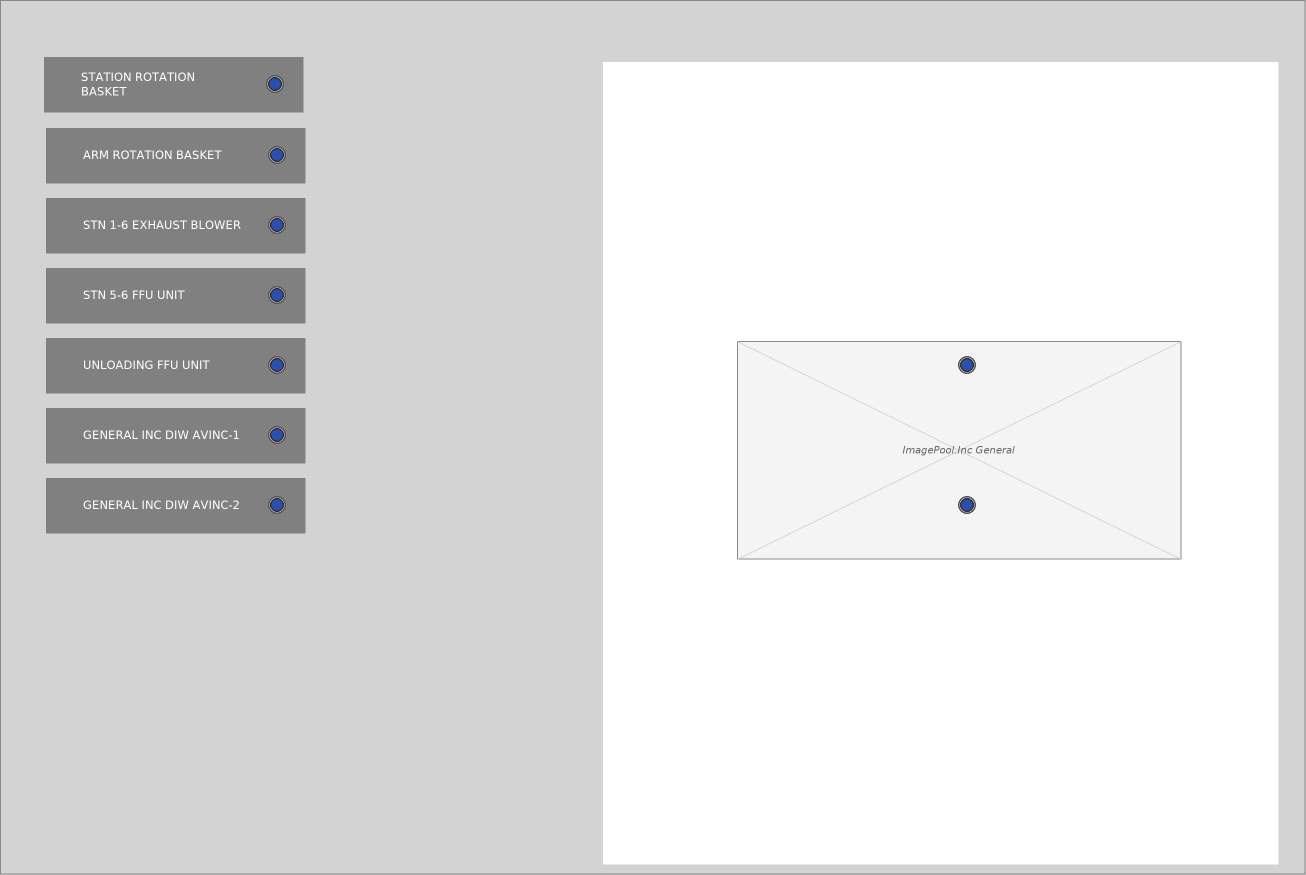
VISUALIZATION Auto_General  // 1306x875
    Rectangle (0,0 1306x875)
    Rectangle (603,62 675x802)
    RoundedRectangle (44,57 259x55)
    Label (78,71 176x27), "STATION ROTATION BASKET"
    Lamp1 (265,74 20x20), variable: ARdsMAP_HmiVariableGeneral.bStnRotationRotaryBarrel_IND, style: Lamp-Lamp1-Blue
    RoundedRectangle (46,198 259x55)
    Label (80,217 178x16), "STN 1-6 EXHAUST BLOWER"
    Lamp1 (267,215 20x20), variable: ARdsMAP_HmiVariableGeneral.bExhaustBlower_IND, style: Lamp-Lamp1-Blue
    Image (737,341 444x218), image: ImagePool.Inc General
    RoundedRectangle (46,408 259x55)
    Label (80,427 176x16), "GENERAL INC DIW AVINC-1"
    Lamp1 (267,425 20x20), variable: ARdsMAP_HmiVariableGeneral.bGeneralIncValve01_IND, style: Lamp-Lamp1-Blue
    RoundedRectangle (46,478 259x55)
    Label (80,497 178x16), "GENERAL INC DIW AVINC-2"
    Lamp1 (267,495 20x20), variable: ARdsMAP_HmiVariableGeneral.bGeneralIncValve02_IND, style: Lamp-Lamp1-Blue
    RoundedRectangle (46,128 259x55)
    Label (80,147 176x16), "ARM ROTATION BASKET"
    Lamp1 (267,145 20x20), variable: ARdsMAP_HmiVariableGeneral.bRobotRotationRotaryBarrel_IND, style: Lamp-Lamp1-Blue
    Lamp1 (957,355 20x20), variable: ARdsMAP_HmiVariableGeneral.bGeneralIncValve01_IND, style: Lamp-Lamp1-Blue
    Lamp1 (957,495 20x20), variable: ARdsMAP_HmiVariableGeneral.bGeneralIncValve02_IND, style: Lamp-Lamp1-Blue
    RoundedRectangle (46,268 259x55)
    Label (80,287 178x16), "STN 5-6 FFU UNIT"
    Lamp1 (267,285 20x20), variable: ARdsMAP_HmiVariableGeneral.bFFU01_IND, style: Lamp-Lamp1-Blue
    RoundedRectangle (46,338 259x55)
    Label (80,357 178x16), "UNLOADING FFU UNIT"
    Lamp1 (267,355 20x20), variable: ARdsMAP_HmiVariableGeneral.bFFU02_IND, style: Lamp-Lamp1-Blue
END_VISUALIZATION

(* stored: Version 1.1.0.1, ProductVersion 3.1.4024.12
   Visu Auto_General: Id {d2faa635-4892-437a-82ed-622115d7b6a8} *)
